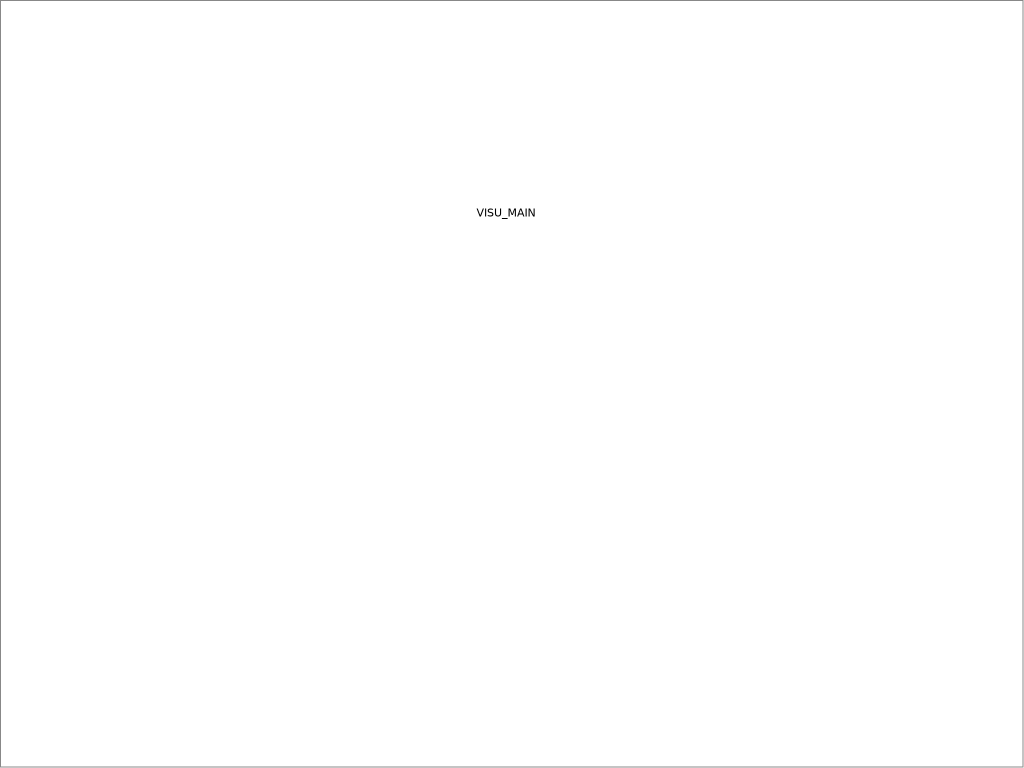
VISUALIZATION visu_main  // 1024x768
    Label (431,198 150x30), "VISU_MAIN"
END_VISUALIZATION

(* stored: Version 1.1.0.1, ProductVersion 3.1.4024.12
   Visu visu_main: Id {c7667e47-18d6-49d4-8b1c-6249f0c3ef26} *)
